FUNCTION_BLOCK InterfaceControlV2
VAR_INPUT
	pbGreen : BOOL; //start
	pbRed : BOOL;	//stop
	pbYellow: BOOL; //error reset
	
	commStart AT%M* : BOOL;
	commStop AT%M* : BOOL;
	commErrorReset AT%M* : BOOL;
	commErrorIgnore AT%M* : BOOL;
	commInit AT%M* : BOOL;
	commPurge AT%M* : BOOL;
END_VAR
VAR_OUTPUT
	
	requestPause : BOOL;
	requestResume: BOOL;
	
	requestInit : BOOL;
	requestErrorClear : eErrorClearWays;
	
	requestPurge : BOOL;
		
END_VAR

requestPause := commStop OR pbRed;
requestResume := commStart OR pbGreen;

IF commErrorReset OR pbYellow THEN
	requestErrorClear := eErrorClearWays.RESET;
ELSIF commErrorIgnore THEN
	requestErrorClear := eErrorClearWays.IGNORE;
ELSE 
	//default
	requestErrorClear := eErrorClearWays.NO_ACTION;	
END_IF

//Initialization
requestInit := commInit;
//Purge request
requestPurge := commPurge; 
//one-shot control clear 
commStart := FALSE;
commStop := FALSE;
commErrorReset := FALSE;
commErrorIgnore:= FALSE;
commInit:= FALSE;
commPurge := FALSE;

END_FUNCTION_BLOCK

(* stored: Version 1.1.0.1, ProductVersion 3.1.4024.0
   POU InterfaceControlV2: Id {5c9a5b58-14bf-4ff5-afb4-63b993847649}, SpecialFunc None *)
